{attribute 'qualified_only'}
{attribute 'strict'}
TYPE EFeedbackMsgIO :
(
	PositionMsg := 10
);
END_TYPE

(* stored: Version 1.1.0.1, ProductVersion 3.1.4024.12
   DUT EFeedbackMsgIO: Id {8f8b3fa1-2c58-4333-adf4-826cb8f6ad3d} *)
